FUNCTION_BLOCK FB_Sequence IMPLEMENTS I_Sequence
VAR
	iParent:			I_Component;
	nNextNumber:		INT;
	stActual:			ST_Sequence;
	aHistory:			ARRAY [0..Parameters.nSequence] OF ST_Sequence;
	fbTimeout:			TON;
	fbDelay: 			TON;
END_VAR

// https://github.com/PeterZerlauth/Tc3_Component
IF iParent.P_Mode = E_Mode.Manual THEN
	stActual.nNumber:= E_Sequence.Manual;
	stActual.sMessage:= 'Manual';
END_IF

METHOD FB_init : BOOL
VAR_INPUT
	bInitRetains : BOOL; // if TRUE, the retain variables are initialized (warm start / cold start)
	bInCopyCode : BOOL;  // if TRUE, the instance afterwards gets moved into the copy code (online change)
	iParent:			I_Component;
END_VAR
THIS^.iParent:= iParent;
END_METHOD

METHOD PUBLIC M_Await 
VAR_INPUT
	sMessage:				STRING(255);		
	tTimeout:				TIME;
	tDelay:					TIME;	
	bPause:					BOOL;
	bReturn:				BOOL;
	nNumber:				INT;
END_VAR
IF bReturn THEN
	IF tDelay <> T#0S THEN
		fbDelay(IN:= TRUE);
		IF fbDelay.Q THEN
			stActual.nNumber:= nNumber;
			fbDelay(IN:= FALSE);
			IF bPause THEN
				IF iParent.P_Mode = E_Mode.Semiauto THEN
					iParent.M_Request(E_Request.Pause);		
				END_IF
			END_IF	
		END_IF
	ELSE
		stActual.sMessage:= sMessage;
		stActual.nNumber:= nNumber;
		MemCpy(ADR(aHistory[1]), ADR(aHistory[0]), SIZEOF(ST_Sequence) * Parameters.nSequence);
		aHistory[0]:= stActual;
		fbTimeout(IN:= FALSE);
		IF bPause THEN
			IF iParent.P_Mode = E_Mode.Semiauto THEN
				iParent.M_Request(E_Request.Pause);		
			END_IF
		END_IF	
	END_IF		
ELSE
	IF tTimeout <> T#0S THEN
		fbTimeout(IN:= TRUE);
		IF fbTimeout.Q THEN
			iParent.P_Event.M_AddINT(stActual.nNumber);
			iParent.P_Event.M_Stop('Timeout in sequence number %s', 1);
		END_IF
	END_IF
END_IF
END_METHOD

METHOD M_Reset
stActual.nNumber:= E_Sequence.Start;
stActual.sMessage:= 'E_Sequence.Start';
MemCpy(ADR(aHistory[1]), ADR(aHistory[0]), SIZEOF(ST_Sequence) * Parameters.nSequence);
aHistory[0]:= stActual;
fbDelay(IN:= FALSE);
fbTimeout(IN:= FALSE);
END_METHOD

METHOD M_Set
VAR_INPUT
	nNumber:				INT;
END_VAR
stActual.nNumber:= nNumber;
stActual.sMessage:= 'M_Set';
MemCpy(ADR(aHistory[1]), ADR(aHistory[0]), SIZEOF(ST_Sequence) * Parameters.nSequence);
aHistory[0]:= stActual;
fbDelay(IN:= FALSE);
fbTimeout(IN:= FALSE);
END_METHOD

{attribute 'OPC.UA.DA.Property' := '1'}
{attribute 'monitoring' := 'call'}
PROPERTY PUBLIC P_Message : STRING(255)
GET
P_Message:= stActual.sMessage;
END_GET
END_PROPERTY

{attribute 'OPC.UA.DA.Property' := '1'}
{attribute 'monitoring' := 'call'}
PROPERTY PUBLIC P_Number : INT
GET
P_Number:= stActual.nNumber;
END_GET
END_PROPERTY

END_FUNCTION_BLOCK

(* stored: Version 1.1.0.1
   POU FB_Sequence: Id {4b1aa270-5e63-4fbf-b9b1-b64186ed4cc4}, SpecialFunc None
   Method FB_init: Id {9410888f-1e8d-054b-01cb-f8f70c408f51}
   Method M_Await: Id {1bc0e82b-8467-4f35-a54e-996600fba2bc}
   Method M_Reset: Id {4501245b-63d2-4732-9d5e-f656a322de01}
   Method M_Set: Id {1679b774-aff9-0900-1b9f-6b982123f170}
   Property P_Message: Id {449cb871-a246-0a5a-09bf-a919fbfd178f}
   Get Get: Id {38483f3c-0df1-00ca-344c-1ba32b91480e}
   Property P_Number: Id {3cc751bf-6092-4aa8-8de5-3276200b64ad}
   Get Get: Id {92b3a1f5-52d3-44fe-8629-e1295a1ef489} *)
